(* PLC project Unnamed, Unknown Unnamed 1 *)
(* stored: creationDateTime 2021-05-11T15:41:27, modificationDateTime 2022-01-21T16:47:01 *)

FUNCTION LOOK_UP : REAL
  VAR_INPUT
    IN : REAL;
    S1 : REAL;
    S2 : REAL;
    S3 : REAL;
    Y1 : REAL;
    Y2 : REAL;
    Y3 : REAL;
  END_VAR
  VAR
    SEL0 : INT := 0;
    SEL1 : INT := 1;
    SEL2 : INT := 2;
    SEL3 : INT := 3;
  END_VAR
  VAR  (* added by the conversion: wires and edge detectors of the diagram *)
    _LT6_OUT : BOOL;
    _LT7_OUT : BOOL;
    _ADD23_OUT : INT;
    _MUX24_OUT : REAL;
    _MUX25_OUT : REAL;
  END_VAR

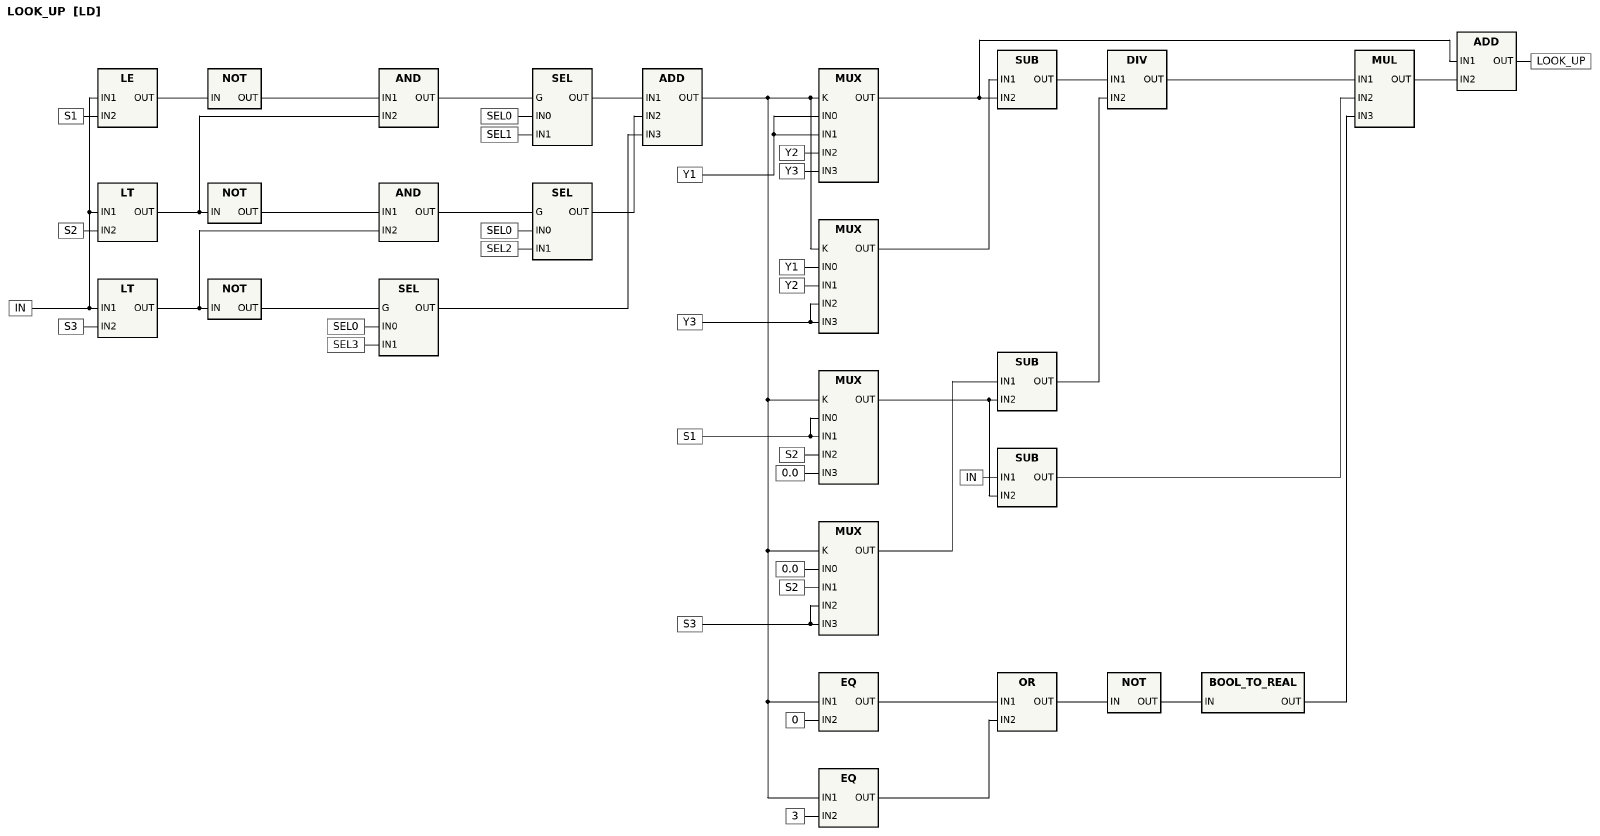
(* LD diagram, written out as Structured Text *)
_LT6_OUT := IN < S2;
_LT7_OUT := IN < S3;
_ADD23_OUT := SEL(NOT (IN <= S1) AND _LT6_OUT, SEL0, SEL1) + SEL(NOT _LT6_OUT AND _LT7_OUT, SEL0, SEL2) + SEL(NOT _LT7_OUT, SEL0, SEL3);
_MUX24_OUT := MUX(_ADD23_OUT, Y1, Y1, Y2, Y3);
_MUX25_OUT := MUX(_ADD23_OUT, S1, S1, S2, 0.0);
LOOK_UP := _MUX24_OUT + (MUX(_ADD23_OUT, Y1, Y2, Y3, Y3) - _MUX24_OUT) / (MUX(_ADD23_OUT, 0.0, S2, S3, S3) - _MUX25_OUT) * (IN - _MUX25_OUT) * BOOL_TO_REAL(NOT (_ADD23_OUT = 0 OR _ADD23_OUT = 3));
END_FUNCTION

PROGRAM SG_LV_PLC
  VAR
    TIME_IN AT %MD0 : REAL;
    TIME_OUT AT %MD1 : REAL;
    SG1_LEVEL AT %MD2 : REAL;
    SG2_LEVEL AT %MD3 : REAL;
    RX_POWER AT %MD4 : REAL;
    FW_PUMPSPEED_1 AT %MD5 : REAL;
    FW_PUMPSPEED_2 AT %MD6 : REAL;
    FW_PUMPSPEED_3 AT %MD7 : REAL;
    FW_PUMP_OnOff_1 AT %MD8 : REAL := 1.0;
    FW_PUMP_OnOff_2 AT %MD9 : REAL := 1.0;
    FW_PUMP_OnOff_3 AT %MD10 : REAL := 0.0;
    MANIPIO_CONTROL AT %MD11 : REAL := 0.0;
    KPI AT %MD12 : REAL := 200.0;
    Ti AT %MD13 : REAL := 600.0;
    LOOK_UP_TEST AT %MD14 : REAL;
  END_VAR
  VAR
    INTEGRAL0 : INTEGRAL;
  END_VAR
  VAR  (* added by the conversion: wires and edge detectors of the diagram *)
    _LOOK_UP33_OUT : REAL;
    _MUL7_OUT : REAL;
    _LIMIT18_OUT : ANY;
    _ADD14_OUT : ANY;
    _SEL23_OUT : REAL;
  END_VAR

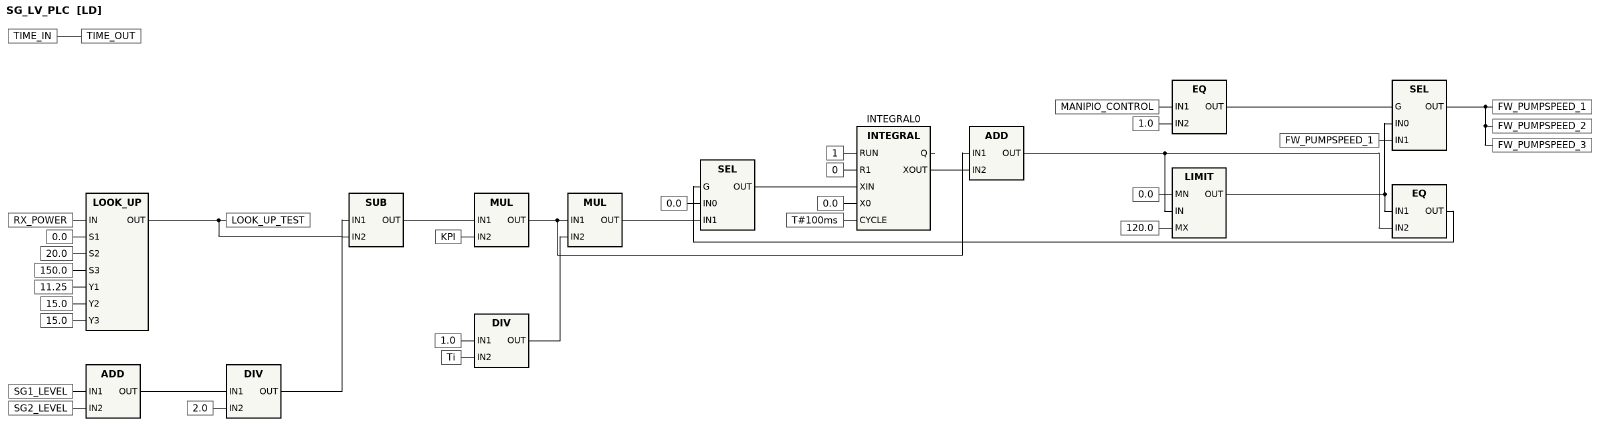
(* LD diagram, written out as Structured Text *)
TIME_OUT := TIME_IN;
_LOOK_UP33_OUT := LOOK_UP(RX_POWER, 0.0, 20.0, 150.0, 11.25, 15.0, 15.0);
_MUL7_OUT := (_LOOK_UP33_OUT - (SG1_LEVEL + SG2_LEVEL) / 2.0) * KPI;
INTEGRAL0(RUN := 1, R1 := 0, XIN := SEL(_LIMIT18_OUT = _ADD14_OUT, 0.0, _MUL7_OUT * (1.0 / Ti)), X0 := 0.0, CYCLE := T#100ms);
_ADD14_OUT := _MUL7_OUT + INTEGRAL0.XOUT;
_LIMIT18_OUT := LIMIT(0.0, _ADD14_OUT, 120.0);
_SEL23_OUT := SEL(MANIPIO_CONTROL = 1.0, _LIMIT18_OUT, FW_PUMPSPEED_1);
FW_PUMPSPEED_1 := _SEL23_OUT;
FW_PUMPSPEED_2 := _SEL23_OUT;
FW_PUMPSPEED_3 := _SEL23_OUT;
LOOK_UP_TEST := _LOOK_UP33_OUT;
END_PROGRAM

CONFIGURATION Config0
  RESOURCE Res0 ON PLC
    TASK task0(INTERVAL := T#100ms, PRIORITY := 0);
    PROGRAM instance0 WITH task0 : SG_LV_PLC;
  END_RESOURCE
END_CONFIGURATION
